INTERFACE I_MotionInterlocks

END_INTERFACE

(* stored: Version 1.1.0.1
   Itf I_MotionInterlocks: Id {7ac89254-d732-4980-b014-871a72f21fa7} *)
